TYPE ST128_Recipe_t :
STRUCT
    xIsTypeMiniOrSmart    : BOOL; // do we have 2 pieces (smart and mini) or just one (others)
END_STRUCT
END_TYPE

(* stored: Version 1.1.0.1, ProductVersion 3.1.4024.6
   DUT ST128_Recipe_t: Id {cfff7e9c-b0c5-46d0-a0ff-b42f6b2382b6} *)
